FUNCTION_BLOCK grab
VAR_INPUT
	 seconds: TIME; //time of moving	  
END_VAR
VAR_OUTPUT
	done: BOOL := FALSE; // output of finished work
END_VAR
VAR
	TimerNewGrab: AUTOtimer;
	activated: BOOL := FALSE; // Internal logic for activation
	grabEnd: BOOL := FALSE;
END_VAR

IF NOT activated THEN
    TimerNewGrab(vrednost := TRUE, inpCas := seconds, outCas => grabEnd);
    activated := TRUE;
END_IF

IF grabEnd  THEN
    TimerNewGrab(vrednost := FALSE, inpCas := seconds, outCas => grabEnd);
	GVL.primi := TRUE;
	GVL.clawWay := FALSE;
    GVL.clawAction := TRUE;  // grab active 
    GVL.grabDone := FALSE; // The move is not finished yet
	GVL.grabMeter := GVL.grabMeter + 0.4;
ELSE
	GVL.primi  := FALSE;
	GVL.clawWay := FALSE;
    GVL.clawAction := FALSE;     // Stop grabing
    GVL.grabDone:= TRUE;  // Mark the end of the move
	activated := FALSE;
END_IF

END_FUNCTION_BLOCK

(* stored: Version 1.1.0.1, ProductVersion 3.1.4024.15
   POU grab: Id {fe9af8bf-9c8d-42eb-8482-49d86b9292ab}, SpecialFunc None *)
